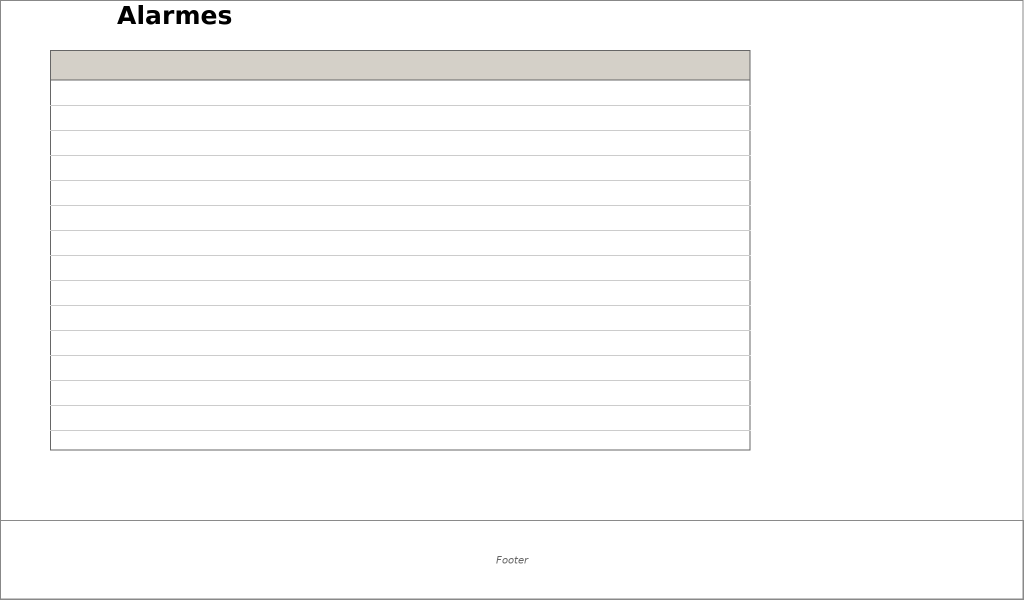
VISUALIZATION Visualization  // 1024x600
    Table (50,50 700x400), data array: prgAlarmHnd.actualEvts
        p3854506369: prgAlarmHnd.actualEvts[INDEX].nSourceID
        p1892666644: prgAlarmHnd.actualEvts[INDEX].nEventID
        p338671338: prgAlarmHnd.actualEvts[INDEX].nClass
        p2170511999: prgAlarmHnd.actualEvts[INDEX].nConfirmState
        p3723444502: prgAlarmHnd.actualEvts[INDEX].nResetState
        p1218418051: prgAlarmHnd.actualEvts[INDEX].sSource
        p746581629: prgAlarmHnd.actualEvts[INDEX].sDate
        p3104783080: prgAlarmHnd.actualEvts[INDEX].sTime
        p2501879983: prgAlarmHnd.actualEvts[INDEX].sComputer
        p7306298: prgAlarmHnd.actualEvts[INDEX].sMessageText
        p1933151965: prgAlarmHnd.actualEvts[INDEX].bQuitMessage
        p3863566920: prgAlarmHnd.actualEvts[INDEX].bConfirmable
        p1755163831: Classe
        p505689113: Origem
        p1757482276: Data
        p4088588272: Hora
        p516019884: Mensagem
        p1014161805: 80 - 1 + INT#1
    Label (100,0 150x30), "Alarmes"
    Frame (0,520 1024x80)
        shows Footer()
END_VISUALIZATION

(* stored: Version 1.1.0.1
   Visu Visualization: Id {fc6abd2a-792d-41c9-817e-7bebd959f874} *)
